FUNCTION_BLOCK FB_Clamp
VAR_INPUT
	
END_VAR
VAR_OUTPUT
END_VAR
VAR
m_csState : CLAMP_STATE;	
m_csStateRequested : CLAMP_STATE;

//Eingänge
m_bIsOpen : BOOL;
m_bIsClosed : BOOL;
m_bIsClosedFull : BOOL;

//Ausgänge
m_bOpen :BOOL;
m_bClose :BOOL;

END_VAR


StateMachine();

METHOD IsClosed : BOOL
VAR_INPUT
END_VAR
IF m_csState = CLAMP_STATE.e_CLOSED THEN
	IsClosed := TRUE;
END_IF
END_METHOD

METHOD IsClosedFull : BOOL
VAR_INPUT
END_VAR
IF m_csState = CLAMP_STATE.e_CLOSED_FULL THEN
	IsClosedFull := TRUE;
END_IF
END_METHOD

METHOD IsError : BOOL
VAR_INPUT
END_VAR
IF m_csState = CLAMP_STATE.e_ERROR THEN
	IsError := TRUE;
END_IF
END_METHOD

METHOD IsOpen : BOOL
VAR_INPUT
END_VAR
IF m_csState = CLAMP_STATE.e_OPEN THEN
	IsOpen := TRUE;
END_IF
END_METHOD

METHOD SetCloseClampEmpty : BOOL
VAR_INPUT
END_VAR
m_csStateRequested := CLAMP_STATE.e_CLOSED;
m_bClose := TRUE;
SetCloseClampEmpty:=TRUE;
END_METHOD

METHOD SetCloseClampFull : BOOL
VAR_INPUT
END_VAR
m_csStateRequested := CLAMP_STATE.e_CLOSED_FULL;
m_bClose := TRUE;
SetCloseClampFull := TRUE;
END_METHOD

METHOD SetOpenClamp : BOOL
VAR_INPUT
END_VAR
m_bOpen := TRUE;
END_METHOD

METHOD StateMachine : BOOL
VAR_INPUT
END_VAR

//m_bIsOpen : BOOL;
//m_bIsClosed : BOOL;
//m_bIsClosedFull : BOOL;

CASE m_csState  OF
	
	CLAMP_STATE.e_OPEN:	
		

		IF m_bIsClosed THEN
			m_csState := CLAMP_STATE.e_CLOSED;		
		END_IF
		
		IF m_bIsClosedFull THEN
			m_csState := CLAMP_STATE.e_CLOSED_FULL;		
		END_IF
		
 	CLAMP_STATE.e_CLOSED_FULL:
	// Fehler wenn falscher Zustand
 		IF m_csStateRequested = CLAMP_STATE.e_CLOSED THEN
  			m_csState := CLAMP_STATE.e_ERROR;
		END_IF
		
		
		IF m_bIsOpen THEN
			m_csState := CLAMP_STATE.e_OPEN;		
		END_IF
	
	CLAMP_STATE.e_CLOSED:
			// Fehler wenn falscher Zustand in diesem Fall: Werkstück erwartet aber nicht im Halter
 		IF m_csStateRequested = CLAMP_STATE.e_CLOSED_FULL THEN
  			m_csState := CLAMP_STATE.e_ERROR;
		END_IF
	
	
		IF m_bIsOpen THEN
			m_csState := CLAMP_STATE.e_OPEN;		
		END_IF
		
CLAMP_STATE.e_ERROR:
		
END_CASE
END_METHOD

END_FUNCTION_BLOCK

(* stored: Version 1.1.0.1, ProductVersion 3.1.4024.0
   POU FB_Clamp: Id {e1c73d33-f6c1-43d7-bcc1-6a1542cba2b5}, SpecialFunc None
   Method IsClosed: Id {f36a093d-e703-4c67-adeb-fb50bcb9d8de}
   Method IsClosedFull: Id {eef664de-fb65-43aa-ac40-3e880256493d}
   Method IsError: Id {dab5c067-89e8-4bf9-906a-f6428ee3c84a}
   Method IsOpen: Id {62f697c4-79e4-48a6-96ed-3a9cb1e39daa}
   Method SetCloseClampEmpty: Id {e1f9b516-b57e-40fd-9545-e308aeecc481}
   Method SetCloseClampFull: Id {a0a19ff9-7e84-4af4-852a-1cae099210e9}
   Method SetOpenClamp: Id {2369cdec-8f4b-40ad-a3b8-c6a7d2e46a99}
   Method StateMachine: Id {9cb897b5-ae35-4796-b6a8-f33e6391352e} *)
